(* CODESYS project mobject-graph-plc-pack.library
   Company: mobject
   DefaultNamespace: mobject-graph-plc-pack
   Version: 0.11.0
   Placeholder: mobject-graph-plc-pack
   Author: mobject dev team
   Title: mobject-graph-plc-pack

Project tree, tasks and I/O mapping:
  libraries: mobject-core, 0.3.0 (mobject); mobject-graph, 0.10.0 (mobject); Tc2_Standard, * (Beckhoff Automation GmbH); Tc2_System, * (Beckhoff Automation GmbH); Tc2_Utilities, * (Beckhoff Automation GmbH)
  Datatypes/
    Alias/
      function block _FLOAT [ST]: FB_init, SetBaseDatatypeReference, Address, ClearReference, Clone, Identifier, MakeReferenceTo, Size, TryMakeReferenceTo, Value
      function block _HRESULT [ST]: FB_init, SetBaseDatatypeReference, Address, ClearReference, Clone, Identifier, MakeReferenceTo, Size, TryMakeReferenceTo, Value
    Enums/
      function block _E_TcEventClass [ST]: FB_init, AddLocalEnumeration, IsEnumeratorValueEqual, SetBaseDatatypeReference, Address, ClearReference, Clone, Identifier, MakeReferenceTo, Size, TryMakeReferenceTo, Value
    Structs/
      function block _TIMESTRUCT [ST]: FB_init, SetMemberReference, Address, ClearReference, Clone, Identifier, MakeReferenceTo, Size, TryMakeReferenceTo, Value, wDay, wDayOfWeek, wHour, wMilliseconds, wMinute, wMonth, wSecond, wYear
    function block PlcDatatypePack [ST]: RegisterWithDatatypes
  Nodes/
    Hardware/
      function block DigitalInputNode [ST]: FB_init, Clone, Dispose, OnExecute
      function block DigitalOutputNode [ST]: FB_init, Clone, Dispose, OnExecute
    function block PlcNodePack [ST]: RegisterWithNodeFactory
  function block PlcPack [ST]: RegisterWithDatatypes, RegisterWithNodeFactory
*)

// Datatypes/Alias/_FLOAT
{attribute 'linkalways'} 
{attribute 'no_explicit_call' := 'This FB is a CLASS and must be accessed using methods or properties'}
{attribute 'enable_dynamic_creation'}
FUNCTION_BLOCK _FLOAT EXTENDS AliasDatatypeBase
VAR
	localData : FLOAT;
	activeData : REFERENCE TO FLOAT REF= localData;
	aliasBaseDatatype : _LREAL(localData);
END_VAR

METHOD FB_init : BOOL
VAR_INPUT
	bInitRetains : BOOL; // if TRUE, the retain variables are initialized (warm start / cold start)
	bInCopyCode : BOOL;  // if TRUE, the instance afterwards gets moved into the copy code (online change)
	InitialValue : FLOAT;
END_VAR
localData := InitialValue;
SetBaseDatatypeReference();
AddBaseDatatype(aliasBaseDatatype);
END_METHOD

METHOD PROTECTED SetBaseDatatypeReference
VAR_INPUT
END_VAR
aliasBaseDatatype.MakeReferenceTo(activeData);
END_METHOD

PROPERTY PUBLIC Address : PVOID
GET
Address := ADR(activeData);
END_GET
END_PROPERTY

METHOD PUBLIC ClearReference
VAR_INPUT
END_VAR
activeData REF= localData;
SetBaseDatatypeReference();
END_METHOD

METHOD PUBLIC Clone : I_Datatype
VAR
    pClone : POINTER TO _FLOAT;
END_VAR
pClone := __NEW(_FLOAT(InitialValue := Value));
Clone := pClone^;
END_METHOD

PROPERTY PUBLIC Identifier : T_MAXSTRING
GET
Identifier := 'FLOAT';
END_GET
END_PROPERTY

METHOD PUBLIC MakeReferenceTo
VAR_INPUT
	ReferenceTarget : REFERENCE TO FLOAT;
END_VAR
activeData REF= ReferenceTarget;
SetBaseDatatypeReference();
END_METHOD

PROPERTY PUBLIC Size : UDINT
GET
Size := SIZEOF(activeData);
END_GET
END_PROPERTY

METHOD TryMakeReferenceTo : BOOL
VAR_INPUT
	Target : I_Datatype;
END_VAR
VAR
	targetAsAlias : I_AliasDatatype;
	pTargetData : POINTER TO FLOAT;
END_VAR
IF NOT Target.TryResolveAsAliasDatatype(targetAsAlias) THEN
	RETURN;
END_IF

IF targetAsAlias.Identifier <> Identifier THEN
	RETURN;
END_IF

pTargetData := Target.Address;
activeData REF= pTargetData^;
SetBaseDatatypeReference();
TryMakeReferenceTo := TRUE;
END_METHOD

PROPERTY PUBLIC Value : REFERENCE TO FLOAT
GET
Value REF= activeData;
END_GET
END_PROPERTY

END_FUNCTION_BLOCK

// Datatypes/Alias/_HRESULT
{attribute 'linkalways'} 
{attribute 'no_explicit_call' := 'This FB is a CLASS and must be accessed using methods or properties'}
{attribute 'enable_dynamic_creation'}
FUNCTION_BLOCK _HRESULT EXTENDS AliasDatatypeBase
VAR
	localData : HRESULT;
	activeData : REFERENCE TO HRESULT REF= localData;
	aliasBaseDatatype : _DINT(localData);
END_VAR

METHOD FB_init : BOOL
VAR_INPUT
	bInitRetains : BOOL; // if TRUE, the retain variables are initialized (warm start / cold start)
	bInCopyCode : BOOL;  // if TRUE, the instance afterwards gets moved into the copy code (online change)
	InitialValue : HRESULT;
END_VAR
localData := InitialValue;
SetBaseDatatypeReference();
AddBaseDatatype(aliasBaseDatatype);
END_METHOD

METHOD PROTECTED SetBaseDatatypeReference
VAR_INPUT
END_VAR
aliasBaseDatatype.MakeReferenceTo(activeData);
END_METHOD

PROPERTY PUBLIC Address : PVOID
GET
Address := ADR(activeData);
END_GET
END_PROPERTY

METHOD PUBLIC ClearReference
VAR_INPUT
END_VAR
activeData REF= localData;
SetBaseDatatypeReference();
END_METHOD

METHOD PUBLIC Clone : I_Datatype
VAR
    pClone : POINTER TO _HRESULT;
END_VAR
pClone := __NEW(_HRESULT(InitialValue := Value));
Clone := pClone^;
END_METHOD

PROPERTY PUBLIC Identifier : T_MAXSTRING
GET
Identifier := 'HRESULT';
END_GET
END_PROPERTY

METHOD PUBLIC MakeReferenceTo
VAR_INPUT
	ReferenceTarget : REFERENCE TO HRESULT;
END_VAR
activeData REF= ReferenceTarget;
SetBaseDatatypeReference();
END_METHOD

PROPERTY PUBLIC Size : UDINT
GET
Size := SIZEOF(activeData);
END_GET
END_PROPERTY

METHOD TryMakeReferenceTo : BOOL
VAR_INPUT
	Target : I_Datatype;
END_VAR
VAR
	targetAsAlias : I_AliasDatatype;
	pTargetData : POINTER TO HRESULT;
END_VAR
IF NOT Target.TryResolveAsAliasDatatype(targetAsAlias) THEN
	RETURN;
END_IF

IF targetAsAlias.Identifier <> Identifier THEN
	RETURN;
END_IF

pTargetData := Target.Address;
activeData REF= pTargetData^;
SetBaseDatatypeReference();
TryMakeReferenceTo := TRUE;
END_METHOD

PROPERTY PUBLIC Value : REFERENCE TO HRESULT
GET
Value REF= activeData;
END_GET
END_PROPERTY

END_FUNCTION_BLOCK

// Datatypes/Enums/_E_TcEventClass
{attribute 'linkalways'} 
{attribute 'no_explicit_call' := 'This FB is a CLASS and must be accessed using methods or properties'}
{attribute 'enable_dynamic_creation'}
FUNCTION_BLOCK _E_TcEventClass EXTENDS EnumDatatypeBase
VAR
	localData : E_TcEventClass;
	activeData : REFERENCE TO E_TcEventClass;
	enumBaseDatatype : _UINT(localData);
END_VAR

METHOD FB_init : BOOL
VAR_INPUT
	bInitRetains : BOOL; // if TRUE, the retain variables are initialized (warm start / cold start)
	bInCopyCode : BOOL;  // if TRUE, the instance afterwards gets moved into the copy code (online change)
	InitialValue : E_TcEventClass;
END_VAR
localData := InitialValue;
AddBaseDatatype(enumBaseDatatype);
ClearReference();

AddLocalEnumeration('TCEVENTCLASS_NONE', E_TcEventClass.TCEVENTCLASS_NONE);
AddLocalEnumeration('TCEVENTCLASS_MAINTENANCE', E_TcEventClass.TCEVENTCLASS_MAINTENANCE);
AddLocalEnumeration('TCEVENTCLASS_MESSAGE', E_TcEventClass.TCEVENTCLASS_MESSAGE);
AddLocalEnumeration('TCEVENTCLASS_HINT', E_TcEventClass.TCEVENTCLASS_HINT);
AddLocalEnumeration('TCEVENTCLASS_STATEINFO', E_TcEventClass.TCEVENTCLASS_STATEINFO);
AddLocalEnumeration('TCEVENTCLASS_INSTRUCTION', E_TcEventClass.TCEVENTCLASS_INSTRUCTION);
AddLocalEnumeration('TCEVENTCLASS_WARNING', E_TcEventClass.TCEVENTCLASS_WARNING);
AddLocalEnumeration('TCEVENTCLASS_ALARM', E_TcEventClass.TCEVENTCLASS_ALARM);
AddLocalEnumeration('TCEVENTCLASS_PARAMERROR', E_TcEventClass.TCEVENTCLASS_PARAMERROR);
END_METHOD

METHOD PRIVATE AddLocalEnumeration
VAR_INPUT
	Enumeration : T_MAXSTRING;
	Value : E_TcEventClass;
END_VAR
AddEnumeration(Enumeration, Value);
END_METHOD

METHOD IsEnumeratorValueEqual : BOOL
VAR_INPUT
	Enumerator : I_KeyValueForwardEnumerator;
END_VAR
VAR
	storedValue : E_TcEventClass;
END_VAR
IF NOT Enumerator.TryGet(storedValue) THEN
	RETURN;
END_IF

IsEnumeratorValueEqual := storedValue = activeData;
END_METHOD

METHOD PROTECTED SetBaseDatatypeReference
VAR_INPUT
END_VAR
enumBaseDatatype.MakeReferenceTo(activeData);
END_METHOD

PROPERTY PUBLIC Address : PVOID
GET
Address := ADR(activeData);
END_GET
END_PROPERTY

METHOD PUBLIC ClearReference
VAR_INPUT
END_VAR
activeData REF= localData;
SetBaseDatatypeReference();
END_METHOD

METHOD PUBLIC Clone : I_Datatype
VAR
    pClone : POINTER TO _E_TcEventClass;
END_VAR
pClone := __NEW(_E_TcEventClass(InitialValue := Value));
Clone := pClone^;
END_METHOD

PROPERTY PUBLIC Identifier : T_MAXSTRING
GET
Identifier := 'E_TcEventClass';
END_GET
END_PROPERTY

METHOD PUBLIC MakeReferenceTo
VAR_INPUT
	ReferenceTarget : REFERENCE TO E_TcEventClass;
END_VAR
activeData REF= ReferenceTarget;
SetBaseDatatypeReference();
END_METHOD

PROPERTY PUBLIC Size : UDINT
GET
Size := SIZEOF(activeData);
END_GET
END_PROPERTY

METHOD TryMakeReferenceTo : BOOL
VAR_INPUT
	Target : I_Datatype;
END_VAR
VAR
	targetAsEnum : I_EnumDatatype;
	pTargetData : POINTER TO E_TcEventClass;
END_VAR
IF NOT Target.TryResolveAsEnumDatatype(targetAsEnum) THEN
	RETURN;
END_IF

IF targetAsEnum.Identifier <> Identifier THEN
	RETURN;
END_IF

pTargetData := Target.Address;
activeData REF= pTargetData^;
SetBaseDatatypeReference();
TryMakeReferenceTo := TRUE;
END_METHOD

PROPERTY PUBLIC Value : REFERENCE TO E_TcEventClass
GET
Value REF= activeData;
END_GET
END_PROPERTY

END_FUNCTION_BLOCK

// Datatypes/Structs/_TIMESTRUCT
{attribute 'linkalways'} 
{attribute 'no_explicit_call' := 'This FB is a CLASS and must be accessed using methods or properties'}
{attribute 'enable_dynamic_creation'}
FUNCTION_BLOCK _TIMESTRUCT EXTENDS StructuredDatatypeBase
VAR
	localData : TIMESTRUCT;
	activeData : REFERENCE TO TIMESTRUCT REF= localData;
	_wYear : _WORD(localData.wYear);
	_wMonth : _WORD(localData.wMonth);
	_wDayOfWeek : _WORD(localData.wDayOfWeek);
	_wDay : _WORD(localData.wDay);
	_wHour : _WORD(localData.wHour);
	_wMinute : _WORD(localData.wMinute);
	_wSecond : _WORD(localData.wSecond);
	_wMilliseconds : _WORD(localData.wMilliseconds);
END_VAR

METHOD FB_init : BOOL
VAR_INPUT
	bInitRetains : BOOL; // if TRUE, the retain variables are initialized (warm start / cold start)
	bInCopyCode : BOOL;  // if TRUE, the instance afterwards gets moved into the copy code (online change)
END_VAR
SetMemberReference();
AddMember('wYear',_wYear);
AddMember('wMonth',_wMonth);
AddMember('wDayOfWeek',_wDayOfWeek);
AddMember('wDay',_wDay);
AddMember('wHour',_wHour);
AddMember('wMinute',_wMinute);
AddMember('wSecond',_wSecond);
AddMember('wMilliseconds',_wMilliseconds);
END_METHOD

METHOD PROTECTED SetMemberReference
VAR_INPUT
END_VAR
_wYear.MakeReferenceTo(activeData.wYear);
_wMonth.MakeReferenceTo(activeData.wMonth);
_wDayOfWeek.MakeReferenceTo(activeData.wDayOfWeek);
_wDay.MakeReferenceTo(activeData.wDay);
_wHour.MakeReferenceTo(activeData.wHour);
_wMinute.MakeReferenceTo(activeData.wMinute);
_wSecond.MakeReferenceTo(activeData.wSecond);
_wMilliseconds.MakeReferenceTo(activeData.wMilliseconds);
END_METHOD

PROPERTY PUBLIC Address : PVOID
GET
Address := ADR(activeData);
END_GET
END_PROPERTY

METHOD PUBLIC ClearReference
VAR_INPUT
END_VAR
activeData REF= localData;
SetMemberReference();
END_METHOD

METHOD PUBLIC Clone : I_Datatype
VAR
    pClone : POINTER TO _TIMESTRUCT;
END_VAR
pClone := __NEW(_TIMESTRUCT());
pClone^.Value := Value;
Clone := pClone^;
END_METHOD

PROPERTY PUBLIC Identifier : T_MAXSTRING
GET
Identifier := 'TIMESTRUCT';
END_GET
END_PROPERTY

METHOD PUBLIC MakeReferenceTo
VAR_INPUT
	ReferenceTarget : REFERENCE TO TIMESTRUCT;
END_VAR
activeData REF= ReferenceTarget;
SetMemberReference();
END_METHOD

PROPERTY PUBLIC Size : UDINT
GET
Size := SIZEOF(activeData);
END_GET
END_PROPERTY

METHOD TryMakeReferenceTo : BOOL
VAR_INPUT
	Target : I_Datatype;
END_VAR
VAR
	pTargetData : POINTER TO TIMESTRUCT;
END_VAR
IF NOT (Target.TypeName = TypeName) THEN
	RETURN;
END_IF

pTargetData := Target.Address;
activeData REF= pTargetData^;
SetMemberReference();
TryMakeReferenceTo := TRUE;
END_METHOD

PROPERTY PUBLIC Value : REFERENCE TO TIMESTRUCT
GET
Value REF= activeData;
END_GET
END_PROPERTY

PROPERTY PUBLIC wDay : Reference to _WORD
GET
wDay REF= _wDay;
END_GET
END_PROPERTY

PROPERTY PUBLIC wDayOfWeek : Reference to _WORD
GET
wDayOfWeek REF= _wDayOfWeek;
END_GET
END_PROPERTY

PROPERTY PUBLIC wHour : Reference to _WORD
GET
wHour REF= _wHour;
END_GET
END_PROPERTY

PROPERTY PUBLIC wMilliseconds : Reference to _WORD
GET
wMilliseconds REF= _wMilliseconds;
END_GET
END_PROPERTY

PROPERTY PUBLIC wMinute : Reference to _WORD
GET
wMinute REF= _wMinute;
END_GET
END_PROPERTY

PROPERTY PUBLIC wMonth : Reference to _WORD
GET
wMonth REF= _wMonth;
END_GET
END_PROPERTY

PROPERTY PUBLIC wSecond : Reference to _WORD
GET
wSecond REF= _wSecond;
END_GET
END_PROPERTY

PROPERTY PUBLIC wYear : Reference to _WORD
GET
wYear REF= _wYear;
END_GET
END_PROPERTY

END_FUNCTION_BLOCK

// Datatypes/PlcDatatypePack
{attribute 'linkalways'} 
{attribute 'no_explicit_call' := 'This FB is a CLASS and must be accessed using methods or properties'}
{attribute 'enable_dynamic_creation'}
FUNCTION_BLOCK PlcDatatypePack IMPLEMENTS I_DatatypePack
VAR
	
	// alias
    _float : _FLOAT(0.0);
	_hresult : _HRESULT(0);

	// enums
	_e_TcEventClass : _E_TcEventClass(E_TcEventClass.TCEVENTCLASS_NONE);
	
	// structures
	_timestruct : _TIMESTRUCT();
	
END_VAR

METHOD RegisterWithDatatypes
VAR_INPUT
	Datatypes : I_Datatypes;
END_VAR
// alias
Datatypes.RegisterDatatype(_float);
Datatypes.RegisterDatatype(_hresult);

// enums

Datatypes.RegisterDatatype(_e_TcEventClass);

// structures
Datatypes.RegisterDatatype(_timestruct);
END_METHOD

END_FUNCTION_BLOCK

// Nodes/Hardware/DigitalInputNode
{attribute 'linkalways'} 
{attribute 'no_explicit_call' := 'This FB is a CLASS and must be accessed using methods or properties'}
{attribute 'enable_dynamic_creation'}
FUNCTION_BLOCK FINAL DigitalInputNode EXTENDS Node
VAR
	input AT %I* : BOOL;
	out : _BOOL(FALSE);
END_VAR

METHOD FB_init : BOOL
VAR_INPUT
	bInitRetains : BOOL; // if TRUE, the retain variables are initialized (warm start / cold start)
	bInCopyCode : BOOL;  // if TRUE, the instance afterwards gets moved into the copy code (online change)
END_VAR
AddOutput('out', out);
END_METHOD

METHOD PUBLIC Clone : I_Node
VAR
END_VAR
Clone := this^;
END_METHOD

METHOD Dispose
VAR_INPUT
END_VAR
END_METHOD

METHOD PROTECTED OnExecute : HRESULT
VAR
END_VAR
out.value := input;
END_METHOD

END_FUNCTION_BLOCK

// Nodes/Hardware/DigitalOutputNode
{attribute 'linkalways'} 
{attribute 'no_explicit_call' := 'This FB is a CLASS and must be accessed using methods or properties'}
{attribute 'enable_dynamic_creation'}
FUNCTION_BLOCK FINAL DigitalOutputNode EXTENDS Node
VAR
	output AT %Q* : BOOL;
	in : _BOOL(FALSE);
END_VAR

METHOD FB_init : BOOL
VAR_INPUT
	bInitRetains : BOOL; // if TRUE, the retain variables are initialized (warm start / cold start)
	bInCopyCode : BOOL;  // if TRUE, the instance afterwards gets moved into the copy code (online change)
END_VAR
AddInput('in', in);
END_METHOD

METHOD PUBLIC Clone : I_Node
VAR
END_VAR
Clone := this^;
END_METHOD

METHOD Dispose
VAR_INPUT
END_VAR
END_METHOD

METHOD PROTECTED OnExecute : HRESULT
VAR
END_VAR
output := in.value;
END_METHOD

END_FUNCTION_BLOCK

// Nodes/PlcNodePack
{attribute 'linkalways'} 
{attribute 'no_explicit_call' := 'This FB is a CLASS and must be accessed using methods or properties'}
{attribute 'enable_dynamic_creation'}
FUNCTION_BLOCK PlcNodePack IMPLEMENTS I_NodePack
VAR
END_VAR

METHOD PUBLIC RegisterWithNodeFactory
VAR_INPUT
	NodeFactory : I_NodeFactory;
END_VAR
END_METHOD

END_FUNCTION_BLOCK

// PlcPack
{attribute 'linkalways'} 
{attribute 'no_explicit_call' := 'This FB is a CLASS and must be accessed using methods or properties'}
{attribute 'enable_dynamic_creation'}
FUNCTION_BLOCK PlcPack IMPLEMENTS I_GraphPack
VAR
	plcDatatypePack : PlcDatatypePack;
	plcNodePack : PlcNodePack;
END_VAR

METHOD RegisterWithDatatypes
VAR_INPUT
	Datatypes : I_Datatypes;
END_VAR
plcDatatypePack.RegisterWithDatatypes(Datatypes);
END_METHOD

METHOD PUBLIC RegisterWithNodeFactory
VAR_INPUT
	NodeFactory : I_NodeFactory;
END_VAR
plcNodePack.RegisterWithNodeFactory(NodeFactory);
END_METHOD

END_FUNCTION_BLOCK
